TYPE ST_ITC_Function :
(**************************************************************************************
 * 	Application		:	BoxControl Framework
 *	Revision		:	$Revision: 404529 $
 *	Revision date	:	$Date: 2018-04-23 08:21:38 +0200 (Mo., 23 Apr 2018) $
 *	Last changed by	:	$Author: b7bolm $
 *	URL				:	$URL: http://almscdc.swisslog.com/repo/SWPD/Development/BoxControlFramework/20_Release/trunk/01_Software/BCF/BCF/JumpStart/20_Product/10_App/12_E_Functions/10_Lib/10_Conv/01_DUTs/ST_ITC_Function.TcDUT $
 *
 *	Purpose			:	Function ITC structure
 *
 * ------------------------------------------------------------------------------------
 *	Copyright Swisslog [IP AG], Switzerland. All rights reserved.
 * 
 * ------------------------------------------------------------------------------------
 *	
 * 	Revision History: 
 *
 * 	VERSION			DATE			INITIALS			DESCRIPTION
 *	0.1				01.01.2001		swl					Example
 *
 **************************************************************************************)
STRUCT
	FunctionITC		: ST_ITC_FunctionITC; // ITC function data
	ZoneITC			: ARRAY [1..NUMBER_OF_ZONES_PER_FUNCTION] OF ST_ITC_Zone; // ITC Zone data
	ManualMotion	: ST_ITC_ManualMotion; // Command for manual motion
END_STRUCT
END_TYPE

(* stored: Version 1.1.0.1, ProductVersion 3.1.4022.12
   DUT ST_ITC_Function: Id {6a26b910-ebbb-42d7-ba9f-4ecabeabfb6c} *)
